FUNCTION_BLOCK GreenMasterDI EXTENDS GreenMasterDI_Base
VAR_INPUT
END_VAR
VAR_OUTPUT
END_VAR
VAR
	IO_DI_01: DigitalInput;
	IO_DI_02: DigitalInput;
	IO_DI_03: DigitalInput;
	IO_DI_04: DigitalInput;
	IO_DI_05: DigitalInput;
	IO_DI_06: DigitalInput;
	IO_DI_07: DigitalInput;
	IO_DI_08: DigitalInput;
	IO_DI_09: DigitalInput;
	IO_DI_10: DigitalInput;
	IO_DI_11: DigitalInput;
	IO_DI_12: DigitalInput;
	IO_DI_13: DigitalInput;
	IO_DI_14: DigitalInput;
	IO_DI_15: DigitalInput;
	IO_DI_16: DigitalInput;
	IO_DI_17: DigitalInput;
	IO_DI_18: DigitalInput;
	IO_DI_19: DigitalInput;
	IO_DI_20: DigitalInput;
	IO_DI_21: DigitalInput;
	IO_DI_22: DigitalInput;
	IO_DI_23: DigitalInput;
	IO_DI_24: DigitalInput;
	IO_DI_25: DigitalInput;
	IO_DI_26: DigitalInput;
	IO_DI_27: DigitalInput;
	IO_DI_28: DigitalInput;
	IO_DI_29: DigitalInput;
END_VAR


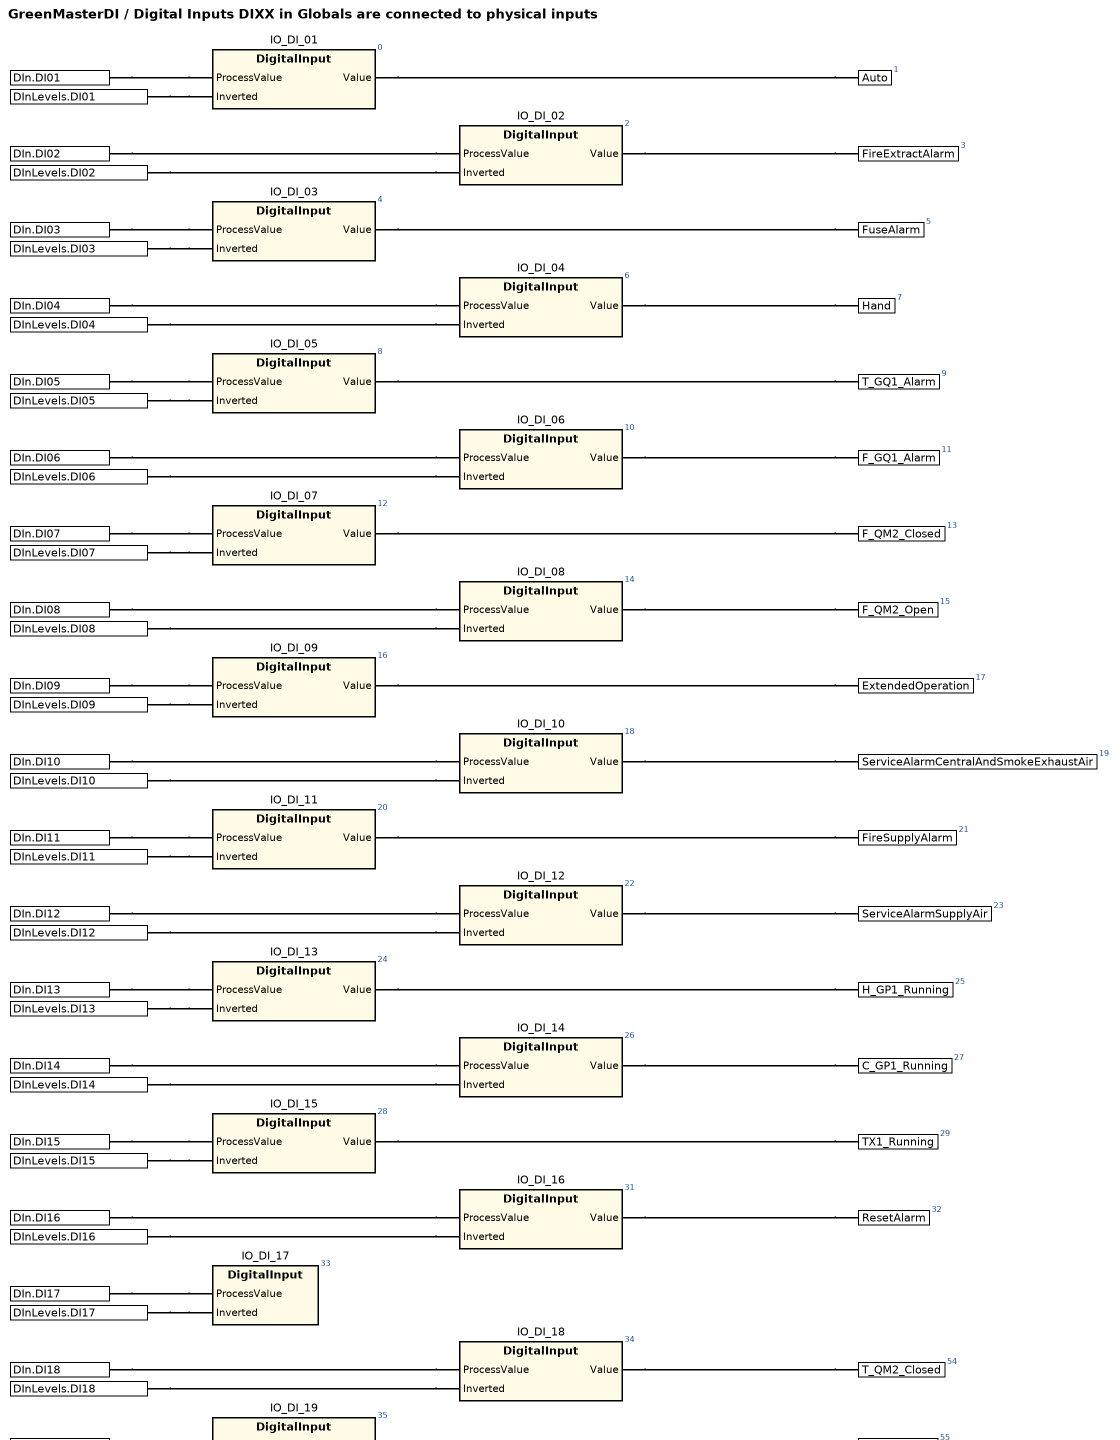
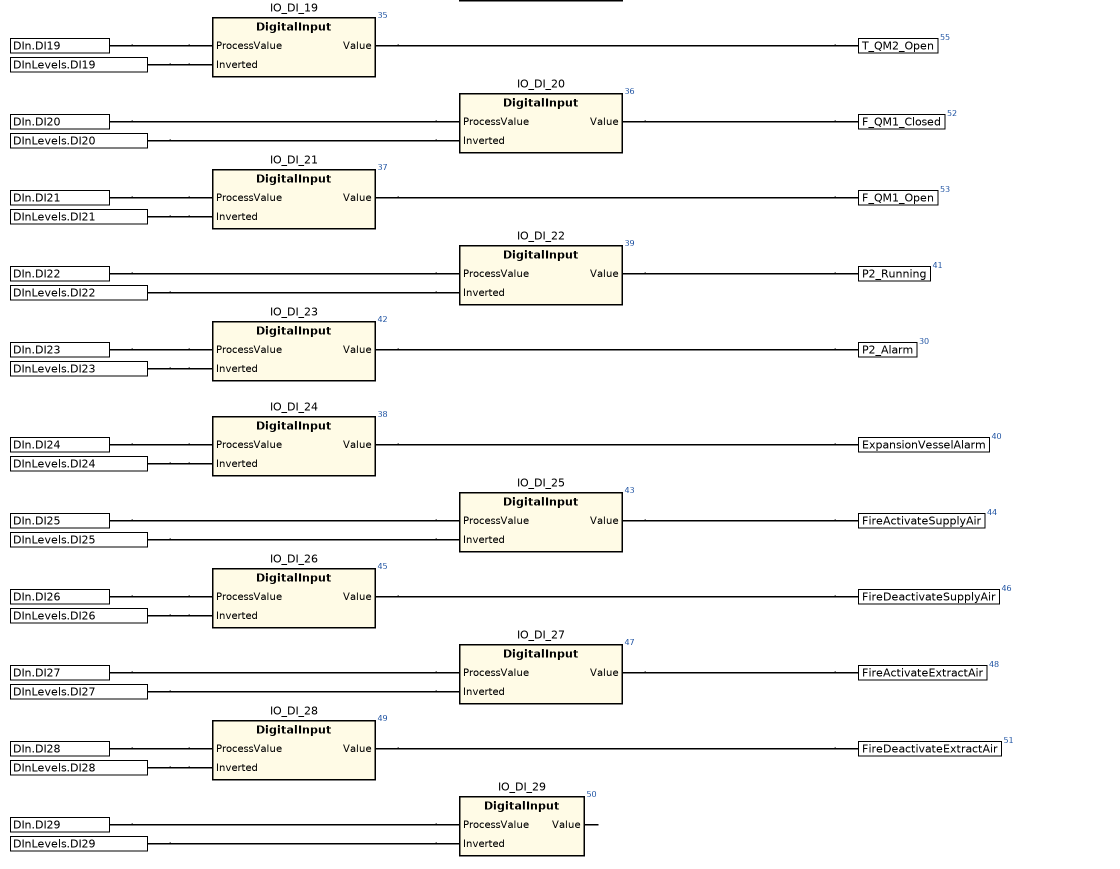
// PAGE Digital Inputs DIXX in Globals are connected to physical inputs
IO_DI_01(ProcessValue := DIn.DI01, Inverted := DInLevels.DI01); // DigitalInput
Auto := IO_DI_01.Value;
IO_DI_02(ProcessValue := DIn.DI02, Inverted := DInLevels.DI02); // DigitalInput
FireExtractAlarm := IO_DI_02.Value;
IO_DI_03(ProcessValue := DIn.DI03, Inverted := DInLevels.DI03); // DigitalInput
FuseAlarm := IO_DI_03.Value;
IO_DI_04(ProcessValue := DIn.DI04, Inverted := DInLevels.DI04); // DigitalInput
Hand := IO_DI_04.Value;
IO_DI_05(ProcessValue := DIn.DI05, Inverted := DInLevels.DI05); // DigitalInput
T_GQ1_Alarm := IO_DI_05.Value;
IO_DI_06(ProcessValue := DIn.DI06, Inverted := DInLevels.DI06); // DigitalInput
F_GQ1_Alarm := IO_DI_06.Value;
IO_DI_07(ProcessValue := DIn.DI07, Inverted := DInLevels.DI07); // DigitalInput
F_QM2_Closed := IO_DI_07.Value;
IO_DI_08(ProcessValue := DIn.DI08, Inverted := DInLevels.DI08); // DigitalInput
F_QM2_Open := IO_DI_08.Value;
IO_DI_09(ProcessValue := DIn.DI09, Inverted := DInLevels.DI09); // DigitalInput
ExtendedOperation := IO_DI_09.Value;
IO_DI_10(ProcessValue := DIn.DI10, Inverted := DInLevels.DI10); // DigitalInput
ServiceAlarmCentralAndSmokeExhaustAir := IO_DI_10.Value;
IO_DI_11(ProcessValue := DIn.DI11, Inverted := DInLevels.DI11); // DigitalInput
FireSupplyAlarm := IO_DI_11.Value;
IO_DI_12(ProcessValue := DIn.DI12, Inverted := DInLevels.DI12); // DigitalInput
ServiceAlarmSupplyAir := IO_DI_12.Value;
IO_DI_13(ProcessValue := DIn.DI13, Inverted := DInLevels.DI13); // DigitalInput
H_GP1_Running := IO_DI_13.Value;
IO_DI_14(ProcessValue := DIn.DI14, Inverted := DInLevels.DI14); // DigitalInput
C_GP1_Running := IO_DI_14.Value;
IO_DI_15(ProcessValue := DIn.DI15, Inverted := DInLevels.DI15); // DigitalInput
TX1_Running := IO_DI_15.Value;
P2_Alarm := IO_DI_23.Value;
IO_DI_16(ProcessValue := DIn.DI16, Inverted := DInLevels.DI16); // DigitalInput
ResetAlarm := IO_DI_16.Value;
IO_DI_17(ProcessValue := DIn.DI17, Inverted := DInLevels.DI17); // DigitalInput
IO_DI_18(ProcessValue := DIn.DI18, Inverted := DInLevels.DI18); // DigitalInput
IO_DI_19(ProcessValue := DIn.DI19, Inverted := DInLevels.DI19); // DigitalInput
IO_DI_20(ProcessValue := DIn.DI20, Inverted := DInLevels.DI20); // DigitalInput
IO_DI_21(ProcessValue := DIn.DI21, Inverted := DInLevels.DI21); // DigitalInput
IO_DI_24(ProcessValue := DIn.DI24, Inverted := DInLevels.DI24); // DigitalInput
IO_DI_22(ProcessValue := DIn.DI22, Inverted := DInLevels.DI22); // DigitalInput
ExpansionVesselAlarm := IO_DI_24.Value;
P2_Running := IO_DI_22.Value;
IO_DI_23(ProcessValue := DIn.DI23, Inverted := DInLevels.DI23); // DigitalInput
IO_DI_25(ProcessValue := DIn.DI25, Inverted := DInLevels.DI25); // DigitalInput
FireActivateSupplyAir := IO_DI_25.Value;
IO_DI_26(ProcessValue := DIn.DI26, Inverted := DInLevels.DI26); // DigitalInput
FireDeactivateSupplyAir := IO_DI_26.Value;
IO_DI_27(ProcessValue := DIn.DI27, Inverted := DInLevels.DI27); // DigitalInput
FireActivateExtractAir := IO_DI_27.Value;
IO_DI_28(ProcessValue := DIn.DI28, Inverted := DInLevels.DI28); // DigitalInput
IO_DI_29(ProcessValue := DIn.DI29, Inverted := DInLevels.DI29); // DigitalInput
FireDeactivateExtractAir := IO_DI_28.Value;
F_QM1_Closed := IO_DI_20.Value;
F_QM1_Open := IO_DI_21.Value;
T_QM2_Closed := IO_DI_18.Value;
T_QM2_Open := IO_DI_19.Value;

END_FUNCTION_BLOCK

(* stored: Version 1.1.0.1, ProductVersion 3.1.4024.6
   POU GreenMasterDI: Id {c4d88455-9985-409d-8af1-319a0d6573ae}, SpecialFunc None *)
